% RSLogix 500 project ANDERSON.RSS, saved by version 11.00.00.00 %
PROJECT "ANDERSON"    % processor: MicroLogix 1000 %

PROGRAM FILES
  LAD 2 "MAIN_PROG"  26 rungs
  LAD 3 "USER_FAULT"  1 rungs
  LAD 4 "HSC_INT"  1 rungs
  LAD 5 "STI_INT"  1 rungs
  LAD 6, 7, 8, 9, 10, 11, 12, 13, 14, 15, 16: only END

DATA FILES
  O0 OUTPUT  1 elements
  I1 INPUT  2 elements
  S2 STATUS  33 elements
  B3 BINARY  32 elements
  T4 TIMER  40 elements
  C5 COUNTER  32 elements
  R6 CONTROL  16 elements
  N7 INTEGER  105 elements

LADDER 2 "MAIN_PROG"
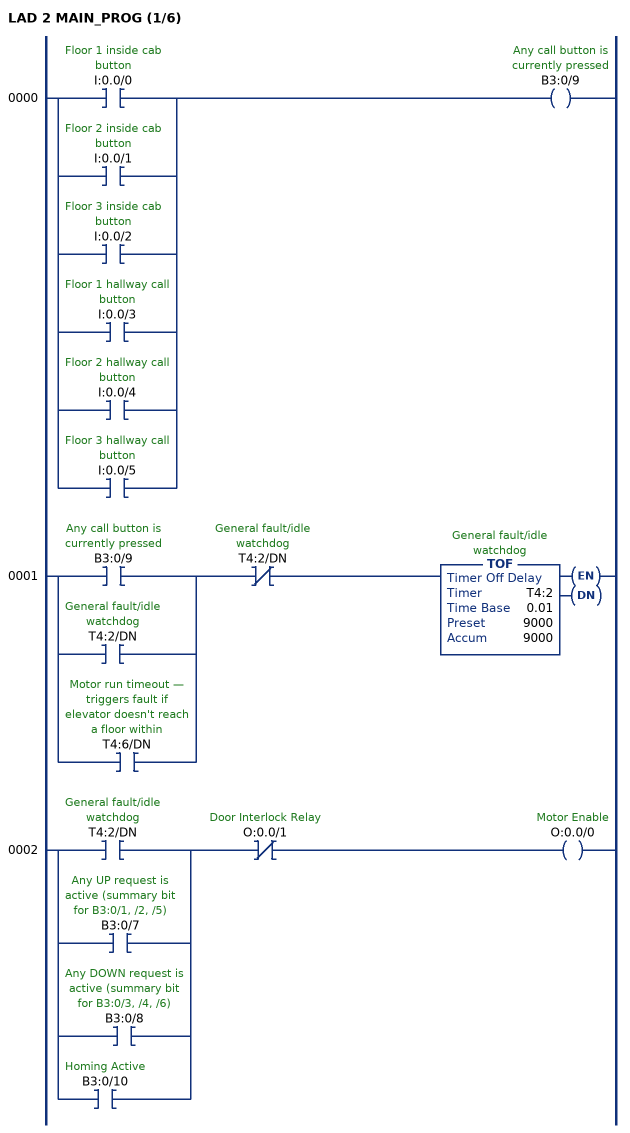
% Rung: 0 %
SOR BST XIC I:0.0/0 NXB XIC I:0.0/1 NXB XIC I:0.0/2 NXB XIC I:0.0/3 NXB XIC I:0.0/4 NXB XIC I:0.0/5 BND OTE B3:0/9 EOR
%   I:0.0/0  "Floor 1 inside cab button" %
%   I:0.0/1  "Floor 2 inside cab button" %
%   I:0.0/2  "Floor 3 inside cab button" %
%   I:0.0/3  "Floor 1 hallway call button" %
%   I:0.0/4  "Floor 2 hallway call button" %
%   I:0.0/5  "Floor 3 hallway call button" %
%   B3:0/9  "Any call button is currently pressed" %
% Rung: 1 %
SOR BST XIC B3:0/9 NXB XIC T4:2/DN NXB XIC T4:6/DN BND XIO T4:2/DN TOF T4:2 0.01 9000 9000 EOR
%   B3:0/9  "Any call button is currently pressed" %
%   T4:2  "General fault/idle watchdog" %
%   T4:6  "Motor run timeout — triggers fault if elevator doesn't reach a floor within" %
% Rung: 2 %
SOR BST XIC T4:2/DN NXB XIC B3:0/7 NXB XIC B3:0/8 NXB XIC B3:0/10 BND XIO O:0.0/1 OTE O:0.0/0 EOR
%   T4:2  "General fault/idle watchdog" %
%   B3:0/7  "Any UP request is active (summary bit for B3:0/1, /2, /5)" %
%   B3:0/8  "Any DOWN request is active (summary bit for B3:0/3, /4, /6)" %
%   B3:0/10  "Homing Active" %
%   O:0.0/1  "Door Interlock Relay" %
%   O:0.0/0  "Motor Enable" %

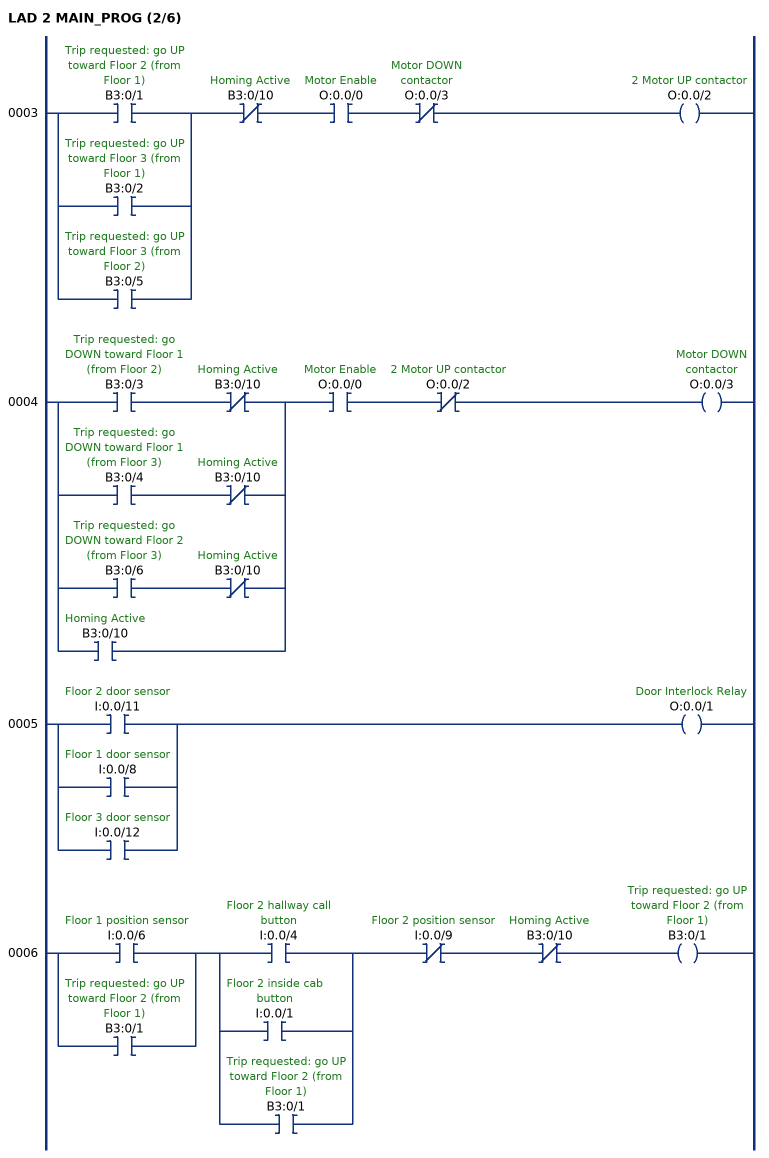
% Rung: 3 %
SOR BST XIC B3:0/1 NXB XIC B3:0/2 NXB XIC B3:0/5 BND XIO B3:0/10 XIC O:0.0/0 XIO O:0.0/3 OTE O:0.0/2 EOR
%   B3:0/1  "Trip requested: go UP toward Floor 2 (from Floor 1)" %
%   B3:0/2  "Trip requested: go UP toward Floor 3 (from Floor 1)" %
%   B3:0/5  "Trip requested: go UP toward Floor 3 (from Floor 2)" %
%   B3:0/10  "Homing Active" %
%   O:0.0/0  "Motor Enable" %
%   O:0.0/3  "Motor DOWN contactor" %
%   O:0.0/2  "2 Motor UP contactor" %
% Rung: 4 %
SOR BST XIC B3:0/3 XIO B3:0/10 NXB XIC B3:0/4 XIO B3:0/10 NXB XIC B3:0/6 XIO B3:0/10 NXB XIC B3:0/10 BND XIC O:0.0/0 XIO O:0.0/2 OTE O:0.0/3 EOR
%   B3:0/3  "Trip requested: go DOWN toward Floor 1 (from Floor 2)" %
%   B3:0/10  "Homing Active" %
%   B3:0/4  "Trip requested: go DOWN toward Floor 1 (from Floor 3)" %
%   B3:0/6  "Trip requested: go DOWN toward Floor 2 (from Floor 3)" %
%   O:0.0/0  "Motor Enable" %
%   O:0.0/2  "2 Motor UP contactor" %
%   O:0.0/3  "Motor DOWN contactor" %
% Rung: 5 %
SOR BST XIC I:0.0/11 NXB XIC I:0.0/8 NXB XIC I:0.0/12 BND OTE O:0.0/1 EOR
%   I:0.0/11  "Floor 2 door sensor" %
%   I:0.0/8  "Floor 1 door sensor" %
%   I:0.0/12  "Floor 3 door sensor" %
%   O:0.0/1  "Door Interlock Relay" %
% Rung: 6 %
SOR BST XIC I:0.0/6 NXB XIC B3:0/1 BND BST XIC I:0.0/4 NXB XIC I:0.0/1 NXB XIC B3:0/1 BND XIO I:0.0/9 XIO B3:0/10 OTE B3:0/1 EOR
%   I:0.0/6  "Floor 1 position sensor" %
%   B3:0/1  "Trip requested: go UP toward Floor 2 (from Floor 1)" %
%   I:0.0/4  "Floor 2 hallway call button" %
%   I:0.0/1  "Floor 2 inside cab button" %
%   I:0.0/9  "Floor 2 position sensor" %
%   B3:0/10  "Homing Active" %

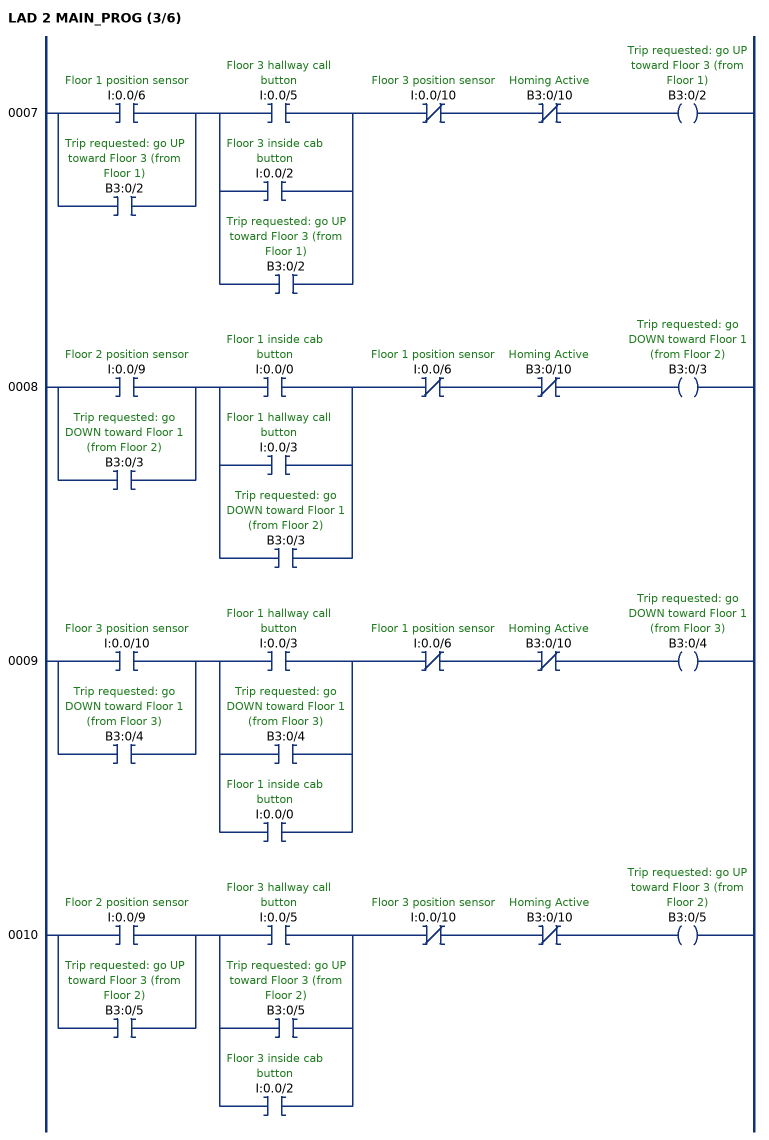
% Rung: 7 %
SOR BST XIC I:0.0/6 NXB XIC B3:0/2 BND BST XIC I:0.0/5 NXB XIC I:0.0/2 NXB XIC B3:0/2 BND XIO I:0.0/10 XIO B3:0/10 OTE B3:0/2 EOR
%   I:0.0/6  "Floor 1 position sensor" %
%   B3:0/2  "Trip requested: go UP toward Floor 3 (from Floor 1)" %
%   I:0.0/5  "Floor 3 hallway call button" %
%   I:0.0/2  "Floor 3 inside cab button" %
%   I:0.0/10  "Floor 3 position sensor" %
%   B3:0/10  "Homing Active" %
% Rung: 8 %
SOR BST XIC I:0.0/9 NXB XIC B3:0/3 BND BST XIC I:0.0/0 NXB XIC I:0.0/3 NXB XIC B3:0/3 BND XIO I:0.0/6 XIO B3:0/10 OTE B3:0/3 EOR
%   I:0.0/9  "Floor 2 position sensor" %
%   B3:0/3  "Trip requested: go DOWN toward Floor 1 (from Floor 2)" %
%   I:0.0/0  "Floor 1 inside cab button" %
%   I:0.0/3  "Floor 1 hallway call button" %
%   I:0.0/6  "Floor 1 position sensor" %
%   B3:0/10  "Homing Active" %
% Rung: 9 %
SOR BST XIC I:0.0/10 NXB XIC B3:0/4 BND BST XIC I:0.0/3 NXB XIC B3:0/4 NXB XIC I:0.0/0 BND XIO I:0.0/6 XIO B3:0/10 OTE B3:0/4 EOR
%   I:0.0/10  "Floor 3 position sensor" %
%   B3:0/4  "Trip requested: go DOWN toward Floor 1 (from Floor 3)" %
%   I:0.0/3  "Floor 1 hallway call button" %
%   I:0.0/0  "Floor 1 inside cab button" %
%   I:0.0/6  "Floor 1 position sensor" %
%   B3:0/10  "Homing Active" %
% Rung: 10 %
SOR BST XIC I:0.0/9 NXB XIC B3:0/5 BND BST XIC I:0.0/5 NXB XIC B3:0/5 NXB XIC I:0.0/2 BND XIO I:0.0/10 XIO B3:0/10 OTE B3:0/5 EOR
%   I:0.0/9  "Floor 2 position sensor" %
%   B3:0/5  "Trip requested: go UP toward Floor 3 (from Floor 2)" %
%   I:0.0/5  "Floor 3 hallway call button" %
%   I:0.0/2  "Floor 3 inside cab button" %
%   I:0.0/10  "Floor 3 position sensor" %
%   B3:0/10  "Homing Active" %

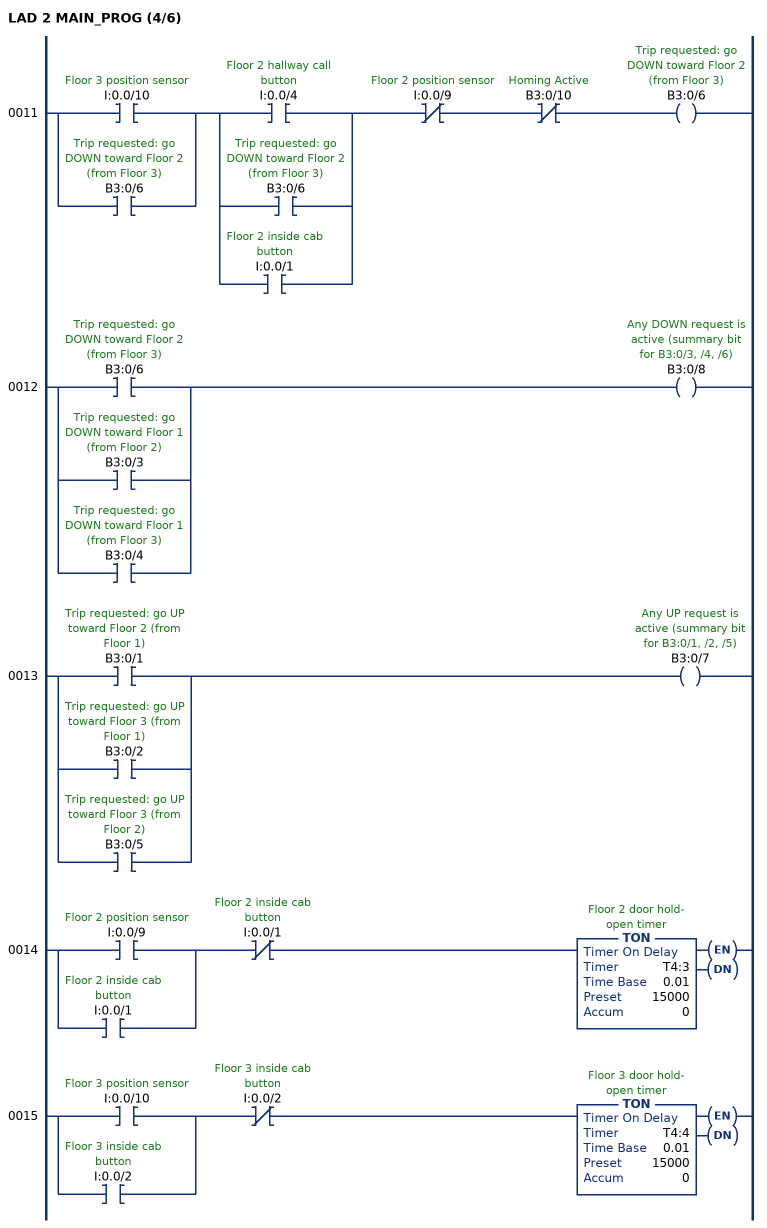
% Rung: 11 %
SOR BST XIC I:0.0/10 NXB XIC B3:0/6 BND BST XIC I:0.0/4 NXB XIC B3:0/6 NXB XIC I:0.0/1 BND XIO I:0.0/9 XIO B3:0/10 OTE B3:0/6 EOR
%   I:0.0/10  "Floor 3 position sensor" %
%   B3:0/6  "Trip requested: go DOWN toward Floor 2 (from Floor 3)" %
%   I:0.0/4  "Floor 2 hallway call button" %
%   I:0.0/1  "Floor 2 inside cab button" %
%   I:0.0/9  "Floor 2 position sensor" %
%   B3:0/10  "Homing Active" %
% Rung: 12 %
SOR BST XIC B3:0/6 NXB XIC B3:0/3 NXB XIC B3:0/4 BND OTE B3:0/8 EOR
%   B3:0/6  "Trip requested: go DOWN toward Floor 2 (from Floor 3)" %
%   B3:0/3  "Trip requested: go DOWN toward Floor 1 (from Floor 2)" %
%   B3:0/4  "Trip requested: go DOWN toward Floor 1 (from Floor 3)" %
%   B3:0/8  "Any DOWN request is active (summary bit for B3:0/3, /4, /6)" %
% Rung: 13 %
SOR BST XIC B3:0/1 NXB XIC B3:0/2 NXB XIC B3:0/5 BND OTE B3:0/7 EOR
%   B3:0/1  "Trip requested: go UP toward Floor 2 (from Floor 1)" %
%   B3:0/2  "Trip requested: go UP toward Floor 3 (from Floor 1)" %
%   B3:0/5  "Trip requested: go UP toward Floor 3 (from Floor 2)" %
%   B3:0/7  "Any UP request is active (summary bit for B3:0/1, /2, /5)" %
% Rung: 14 %
SOR BST XIC I:0.0/9 NXB XIC I:0.0/1 BND XIO I:0.0/1 TON T4:3 0.01 15000 0 EOR
%   I:0.0/9  "Floor 2 position sensor" %
%   I:0.0/1  "Floor 2 inside cab button" %
%   T4:3  "Floor 2 door hold- open timer" %
% Rung: 15 %
SOR BST XIC I:0.0/10 NXB XIC I:0.0/2 BND XIO I:0.0/2 TON T4:4 0.01 15000 0 EOR
%   I:0.0/10  "Floor 3 position sensor" %
%   I:0.0/2  "Floor 3 inside cab button" %
%   T4:4  "Floor 3 door hold- open timer" %

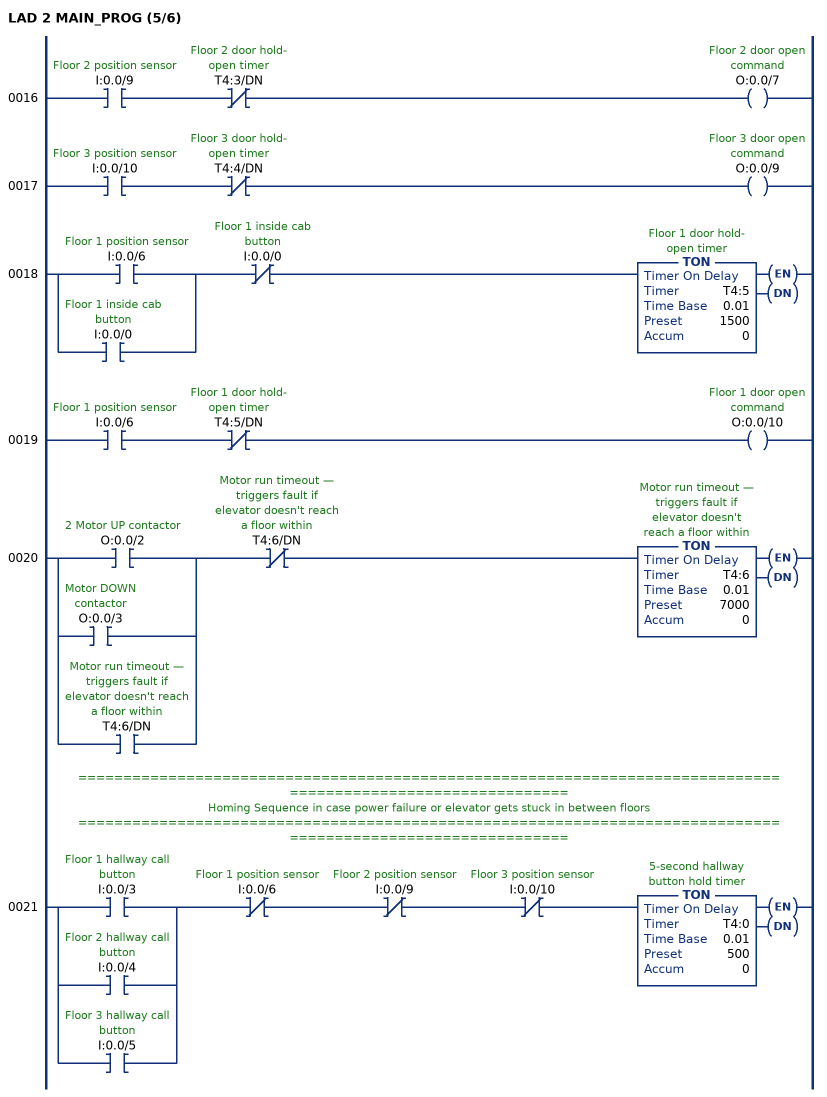
% Rung: 16 %
SOR XIC I:0.0/9 XIO T4:3/DN OTE O:0.0/7 EOR
%   I:0.0/9  "Floor 2 position sensor" %
%   T4:3  "Floor 2 door hold- open timer" %
%   O:0.0/7  "Floor 2 door open command" %
% Rung: 17 %
SOR XIC I:0.0/10 XIO T4:4/DN OTE O:0.0/9 EOR
%   I:0.0/10  "Floor 3 position sensor" %
%   T4:4  "Floor 3 door hold- open timer" %
%   O:0.0/9  "Floor 3 door open command" %
% Rung: 18 %
SOR BST XIC I:0.0/6 NXB XIC I:0.0/0 BND XIO I:0.0/0 TON T4:5 0.01 1500 0 EOR
%   I:0.0/6  "Floor 1 position sensor" %
%   I:0.0/0  "Floor 1 inside cab button" %
%   T4:5  "Floor 1 door hold- open timer" %
% Rung: 19 %
SOR XIC I:0.0/6 XIO T4:5/DN OTE O:0.0/10 EOR
%   I:0.0/6  "Floor 1 position sensor" %
%   T4:5  "Floor 1 door hold- open timer" %
%   O:0.0/10  "Floor 1 door open command" %
% Rung: 20 %
SOR BST XIC O:0.0/2 NXB XIC O:0.0/3 NXB XIC T4:6/DN BND XIO T4:6/DN TON T4:6 0.01 7000 0 EOR
%   O:0.0/2  "2 Motor UP contactor" %
%   O:0.0/3  "Motor DOWN contactor" %
%   T4:6  "Motor run timeout — triggers fault if elevator doesn't reach a floor within" %
% Rung: 21 %
%                                                                                                                                                                                                                                                      =============================================================================================================
% 
%                                                                                                                                                                                                                                                                                            Homing Sequence in case power failure or elevator gets stuck in between floors
% 
% 
%                                                                                                                                                                                                                                                      ============================================================================================================= %
SOR BST XIC I:0.0/3 NXB XIC I:0.0/4 NXB XIC I:0.0/5 BND XIO I:0.0/6 XIO I:0.0/9 XIO I:0.0/10 TON T4:0 0.01 500 0 EOR
%   I:0.0/3  "Floor 1 hallway call button" %
%   I:0.0/4  "Floor 2 hallway call button" %
%   I:0.0/5  "Floor 3 hallway call button" %
%   I:0.0/6  "Floor 1 position sensor" %
%   I:0.0/9  "Floor 2 position sensor" %
%   I:0.0/10  "Floor 3 position sensor" %
%   T4:0  "5-second hallway button hold timer" %

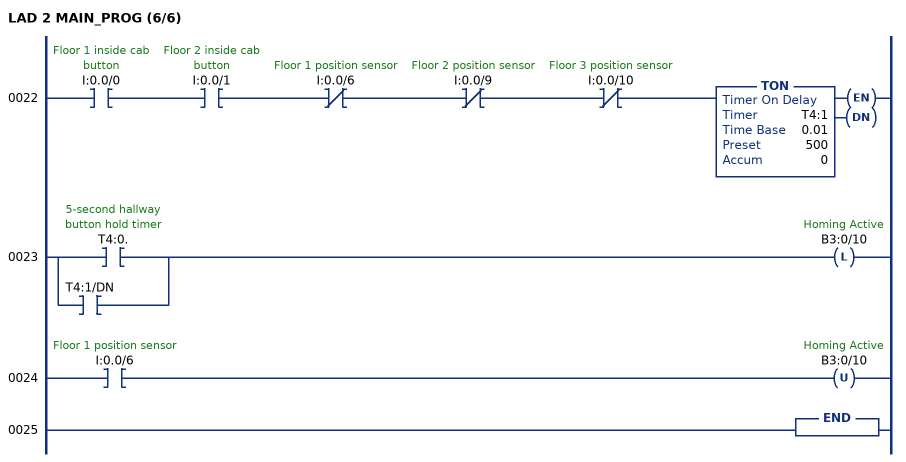
% Rung: 22 %
SOR XIC I:0.0/0 XIC I:0.0/1 XIO I:0.0/6 XIO I:0.0/9 XIO I:0.0/10 TON T4:1 0.01 500 0 EOR
%   I:0.0/0  "Floor 1 inside cab button" %
%   I:0.0/1  "Floor 2 inside cab button" %
%   I:0.0/6  "Floor 1 position sensor" %
%   I:0.0/9  "Floor 2 position sensor" %
%   I:0.0/10  "Floor 3 position sensor" %
% Rung: 23 %
SOR BST XIC T4:0. NXB XIC T4:1/DN BND OTL B3:0/10 EOR
%   T4:0  "5-second hallway button hold timer" %
%   B3:0/10  "Homing Active" %
% Rung: 24 %
SOR XIC I:0.0/6 OTU B3:0/10 EOR
%   I:0.0/6  "Floor 1 position sensor" %
%   B3:0/10  "Homing Active" %
% Rung: 25 %
SOR END EOR

REVISION NOTES
  0: Added Homing sequence

DATA TABLE (non-zero values as saved)
DATA T4
% .PRE .ACC %
% T4:0 % 500 0
% T4:2 % 9000 9000
% T4:3 % 15000 0
% T4:4 % 15000 0
% T4:5 % 1500 0
% T4:6 % 7000 0
